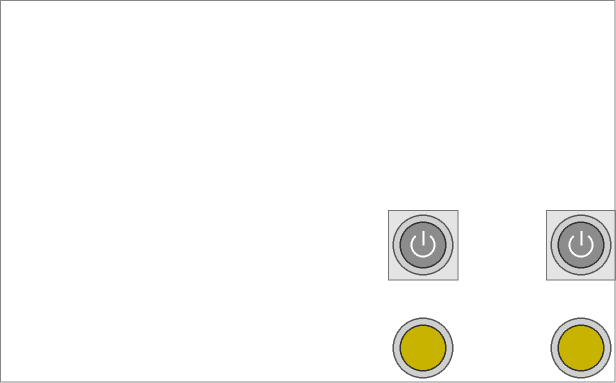
VISUALIZATION Visu  // 616x383
    PowerSwitch (388,210 70x70), variable: MAIN.bS01, behaviour: TOGGLE, style: Switch-PowerSwitch-Gray
    PowerSwitch (546,210 70x70), variable: MAIN.bS02, behaviour: TOGGLE, style: Switch-PowerSwitch-Gray
    Lamp1 (388,313 70x70), variable: MAIN.bQ01, style: Lamp-Lamp1-Yellow
    Lamp1 (546,313 70x70), variable: MAIN.bQ02, style: Lamp-Lamp1-Yellow
END_VISUALIZATION

(* stored: Version 1.1.0.1, ProductVersion 3.1.4024.12
   Visu Visu: Id {bf1ba334-1500-4684-8f78-35772c4c9f30} *)
